// TIA Portal V16 export
// export: Created 2022-09-01T14:27:02.3199962Z, ExportSetting WithDefaults, DisplayName Totally Integrated Automation Portal, DisplayVersion V16, DisplayName TIA Portal Version Control Interface, DisplayVersion V16, DisplayName TIA Portal Openness, DisplayVersion V16, DisplayName STEP 7 Professional, DisplayVersion V16, DisplayName STEP 7 Safety, DisplayVersion V16, DisplayName WinCC Advanced, DisplayVersion V16
FUNCTION "Comando_Avaria_Bombas" : Void   // FC21, LAD
{ S7_Optimized_Access := 'TRUE' }
VERSION : 0.1
// stored: AutoNumber true, IsIECCheckEnabled false, SetENOAutomatically false, UDAEnableTagReadback false
BEGIN

REGION Network 1: Se Bomba 1 Avariar ficam a trabalhar a Bomba 2 e Bomba 3
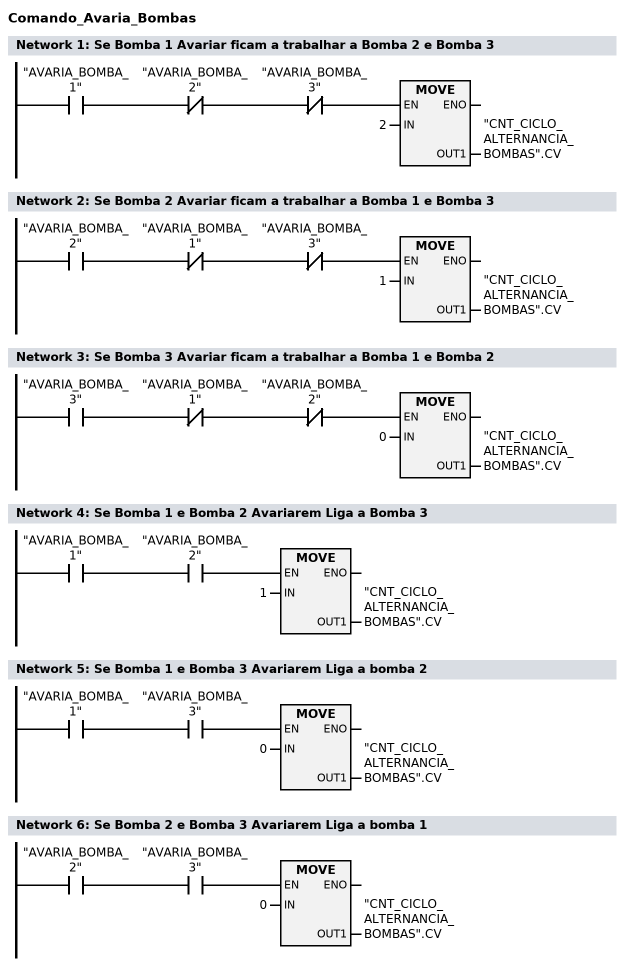
   RUNG wire#powerrail
      Contact( "AVARIA_BOMBA_1" )
      I_Contact( "AVARIA_BOMBA_2" )
      I_Contact( "AVARIA_BOMBA_3" )
      Move(in := 2, out1 => "CNT_CICLO_ALTERNANCIA_BOMBAS".CV)
   END_RUNG
   // the same network as SCL:
   IF "AVARIA_BOMBA_1" AND NOT "AVARIA_BOMBA_2" AND NOT "AVARIA_BOMBA_3" THEN
       "CNT_CICLO_ALTERNANCIA_BOMBAS".CV := 2;
   END_IF;
END_REGION

REGION Network 2: Se Bomba 2 Avariar ficam a trabalhar a Bomba 1 e Bomba 3
   RUNG wire#powerrail
      Contact( "AVARIA_BOMBA_2" )
      I_Contact( "AVARIA_BOMBA_1" )
      I_Contact( "AVARIA_BOMBA_3" )
      Move(in := 1, out1 => "CNT_CICLO_ALTERNANCIA_BOMBAS".CV)
   END_RUNG
   // the same network as SCL:
   IF "AVARIA_BOMBA_2" AND NOT "AVARIA_BOMBA_1" AND NOT "AVARIA_BOMBA_3" THEN
       "CNT_CICLO_ALTERNANCIA_BOMBAS".CV := 1;
   END_IF;
END_REGION

REGION Network 3: Se Bomba 3 Avariar ficam a trabalhar a Bomba 1 e Bomba 2
   RUNG wire#powerrail
      Contact( "AVARIA_BOMBA_3" )
      I_Contact( "AVARIA_BOMBA_1" )
      I_Contact( "AVARIA_BOMBA_2" )
      Move(in := 0, out1 => "CNT_CICLO_ALTERNANCIA_BOMBAS".CV)
   END_RUNG
   // the same network as SCL:
   IF "AVARIA_BOMBA_3" AND NOT "AVARIA_BOMBA_1" AND NOT "AVARIA_BOMBA_2" THEN
       "CNT_CICLO_ALTERNANCIA_BOMBAS".CV := 0;
   END_IF;
END_REGION

REGION Network 4: Se Bomba 1 e Bomba 2 Avariarem Liga a Bomba 3
   RUNG wire#powerrail
      Contact( "AVARIA_BOMBA_1" )
      Contact( "AVARIA_BOMBA_2" )
      Move(in := 1, out1 => "CNT_CICLO_ALTERNANCIA_BOMBAS".CV)
   END_RUNG
   // the same network as SCL:
   IF "AVARIA_BOMBA_1" AND "AVARIA_BOMBA_2" THEN "CNT_CICLO_ALTERNANCIA_BOMBAS".CV := 1; END_IF;
END_REGION

REGION Network 5: Se Bomba 1 e Bomba 3 Avariarem Liga a bomba 2
   RUNG wire#powerrail
      Contact( "AVARIA_BOMBA_1" )
      Contact( "AVARIA_BOMBA_3" )
      Move(in := 0, out1 => "CNT_CICLO_ALTERNANCIA_BOMBAS".CV)
   END_RUNG
   // the same network as SCL:
   IF "AVARIA_BOMBA_1" AND "AVARIA_BOMBA_3" THEN "CNT_CICLO_ALTERNANCIA_BOMBAS".CV := 0; END_IF;
END_REGION

REGION Network 6: Se Bomba 2 e Bomba 3 Avariarem Liga a bomba 1
   RUNG wire#powerrail
      Contact( "AVARIA_BOMBA_2" )
      Contact( "AVARIA_BOMBA_3" )
      Move(in := 0, out1 => "CNT_CICLO_ALTERNANCIA_BOMBAS".CV)
   END_RUNG
   // the same network as SCL:
   IF "AVARIA_BOMBA_2" AND "AVARIA_BOMBA_3" THEN "CNT_CICLO_ALTERNANCIA_BOMBAS".CV := 0; END_IF;
END_REGION
END_FUNCTION
